// TIA Portal V20 export
DATA_BLOCK "BK24"   // DB238
// stored: MemoryReserve 100
   VAR
      "X10-1.SEPA CLAMP TOP REAR UP" : Bool := FALSE;
      "X11-1.SPARE" : Bool := FALSE;
      "X12-1.SEPA CLAMP TOP FRONT UP" : Bool := FALSE;
      "X13-1.SPARE" : Bool := FALSE;
      "X14-1.SEPA CLAMP BTM REAR UP" : Bool := TRUE;
      "X15-1.SPARE" : Bool := FALSE;
      "X16-1.SEPA CLAMP BTM FRONT UP" : Bool := TRUE;
      "X17-1.SPARE" : Bool := FALSE;
      "X10-2.SEPA CLAMP TOP REAR DOWN" : Bool := TRUE;
      "X11-2.SPARE" : Bool := FALSE;
      "X12-2.SEPA CLAMP TOP FRONT DOWN" : Bool := TRUE;
      "X13-2.SPARE" : Bool := FALSE;
      "X14-2.SEPA CLAMP BTM REAR DOWN" : Bool := FALSE;
      "X15-2.SPARE" : Bool := FALSE;
      "X16-2.SEPA CLAMP BTM FRONT DOWN" : Bool := FALSE;
      "X17-2.SPARE" : Bool := FALSE;
   END_VAR
BEGIN
END_DATA_BLOCK
